FUNCTION_BLOCK MoveMoverTask_TestSuite
VAR
	stubAxis : AXIS_REF;
	testMoveTask : MoveToPositionTask := (AxisRef := stubAxis);
	ThisTestSuite : TestSuite<TestSuiteParameter.MaxTestCount>('C:\ProgramData\Beckhoff\TwinCAT\3.1\Boot\MoveMover_Tests.xml') := (TestSuiteName := 'MoveMover Test Suite');
END_VAR

TaskRejectCyclewithNoAxisRefs_Test();
TaskRejectMovewithNoAxisRefs_Test();
TaskRejectsZeroAccelSet_Test();
TaskRejectsZeroVeloMove_Test();
TaskAcceptsValidMoveCommand_Test();
TaskRejectsUnvalidGapSet_Test();
TaskRejectsZeroDecelSet_Test();
TaskRejectsZeroJerkSet_Test();
TaskRejectsDuplicateCall_Test();

METHOD TaskAcceptsValidMoveCommand_Test
VAR_INST
	Expected : BOOL := TRUE;
	Actual	 : BOOL;
END_VAR
IF ThisTestSuite.Test(__POUNAME()).ExecuteTest() THEN
	Actual := SUCCEEDED(testMoveTask.MoveTo(1.0,1.0,tc3_mc3definitions.MC_DIRECTION.mcDirectionNegative,0));
	testMoveTask.Abort();
	ThisTestSuite.Test(__POUNAME()).AssertEqual(Expected, Actual);
END_IF
END_METHOD

METHOD TaskRejectCyclewithNoAxisRefs_Test
VAR_INST
	Expected : BOOL := TRUE;
	Actual	 : BOOL;
END_VAR
IF ThisTestSuite.Test(__POUNAME()).ExecuteTest() THEN
	testMoveTask.AxisRef REF= 16#0;
	Actual := FAILED(testMoveTask.Cycle());
	testMoveTask.AxisRef REF= stubAxis;
	testMoveTask.Abort();
	ThisTestSuite.Test(__POUNAME()).AssertEqual(Expected, Actual);
END_IF
END_METHOD

METHOD TaskRejectMovewithNoAxisRefs_Test
VAR_INST
	Expected : BOOL := TRUE;
	Actual	 : BOOL;
END_VAR
IF ThisTestSuite.Test(__POUNAME()).ExecuteTest() THEN
	testMoveTask.AxisRef REF= 16#0;
	Actual := FAILED(testMoveTask.MoveTo(0.0,0.0,Tc3_Mc3Definitions.MC_DIRECTION.mcDirectionNegative,0));
	testMoveTask.AxisRef REF= stubAxis;
	testMoveTask.Abort();
	ThisTestSuite.Test(__POUNAME()).AssertEqual(Expected, Actual);
END_IF
END_METHOD

METHOD TaskRejectsDuplicateCall_Test : BOOL
VAR_INST
	Expected : BOOL := TRUE;
	Actual	 : BOOL;
END_VAR
IF ThisTestSuite.Test(__POUNAME()).ExecuteTest() THEN
	testMoveTask.MoveTo(1.0,1.0,mc_direction.MC_Positive_Direction,0);
	Actual := SUCCEEDED(testMoveTask.MoveTo(1.0,1.0,tc3_mc3definitions.MC_DIRECTION.mcDirectionNegative,0));
	testMoveTask.Abort();
	ThisTestSuite.Test(__POUNAME()).AssertEqual(Expected, Actual);
END_IF
END_METHOD

METHOD TaskRejectsUnvalidGapSet_Test
VAR_INST
	Expected : BOOL := TRUE;
	Actual	 : BOOL;
END_VAR
IF ThisTestSuite.Test(__POUNAME()).ExecuteTest() THEN
	testMoveTask.Gap := 62.0;
	testMoveTask.Gap := 0.0;
	Actual := testMoveTask.Gap = 62.0;
	ThisTestSuite.Test(__POUNAME()).AssertEqual(Expected, Actual);
END_IF
END_METHOD

METHOD TaskRejectsZeroAccelSet_Test
VAR_INST
	Expected : BOOL := TRUE;
	Actual	 : BOOL;
END_VAR
IF ThisTestSuite.Test(__POUNAME()).ExecuteTest() THEN
	testMoveTask.Acceleration := 32.0;
	testMoveTask.Acceleration := 0.0;
	Actual := testMoveTask.Acceleration = 32.0;
	ThisTestSuite.Test(__POUNAME()).AssertEqual(Expected, Actual);
END_IF
END_METHOD

METHOD TaskRejectsZeroDecelSet_Test
VAR_INST
	Expected : BOOL := TRUE;
	Actual	 : BOOL;
END_VAR
IF ThisTestSuite.Test(__POUNAME()).ExecuteTest() THEN
	testMoveTask.Deceleration := 32.0;
	testMoveTask.Deceleration := 0.0;
	Actual := testMoveTask.Deceleration = 32.0;
	ThisTestSuite.Test(__POUNAME()).AssertEqual(Expected, Actual);
END_IF
END_METHOD

METHOD TaskRejectsZeroJerkSet_Test
VAR_INST
	Expected : BOOL := TRUE;
	Actual	 : BOOL;
END_VAR
IF ThisTestSuite.Test(__POUNAME()).ExecuteTest() THEN
	testMoveTask.Jerk := 32.0;
	testMoveTask.Jerk := 0.0;
	Actual := testMoveTask.Jerk = 32.0;
	ThisTestSuite.Test(__POUNAME()).AssertEqual(Expected, Actual);
END_IF
END_METHOD

METHOD TaskRejectsZeroVeloMove_Test
VAR_INST
	Expected : BOOL := TRUE;
	Actual	 : BOOL;
END_VAR
IF ThisTestSuite.Test(__POUNAME()).ExecuteTest() THEN
	Actual := FAILED(testMoveTask.MoveTo(1.0,0.0,tc3_mc3definitions.MC_DIRECTION.mcDirectionNegative,0));
	testMoveTask.Abort();
	ThisTestSuite.Test(__POUNAME()).AssertEqual(Expected, Actual);
END_IF
END_METHOD

END_FUNCTION_BLOCK

(* stored: Version 1.1.0.1
   POU MoveMoverTask_TestSuite: Id {3c6dc573-70f3-4fa0-a64c-028210806be9}, SpecialFunc None
   Method TaskAcceptsValidMoveCommand_Test: Id {e9d379e6-6863-4b38-8749-39f7f46ba32d}
   Method TaskRejectCyclewithNoAxisRefs_Test: Id {cea8ae0e-65b7-42c7-be1d-83ca270a6f8b}
   Method TaskRejectMovewithNoAxisRefs_Test: Id {936e50d8-e875-4d1c-9c35-f00cbe24977a}
   Method TaskRejectsDuplicateCall_Test: Id {b7f1288f-03aa-4703-8d00-189129abcab9}
   Method TaskRejectsUnvalidGapSet_Test: Id {9434b53d-5dd2-44ed-abe8-7bbd73f61bde}
   Method TaskRejectsZeroAccelSet_Test: Id {0680505a-b3c5-484d-8ec8-d6b7def2f093}
   Method TaskRejectsZeroDecelSet_Test: Id {a9a3bd09-5a19-4b2a-b3d8-3d7c6873a02b}
   Method TaskRejectsZeroJerkSet_Test: Id {d881c961-9d8d-4b46-ae8d-8641b8f61da4}
   Method TaskRejectsZeroVeloMove_Test: Id {23a2a9cd-c0be-4be6-af02-44f166ce64a0} *)
